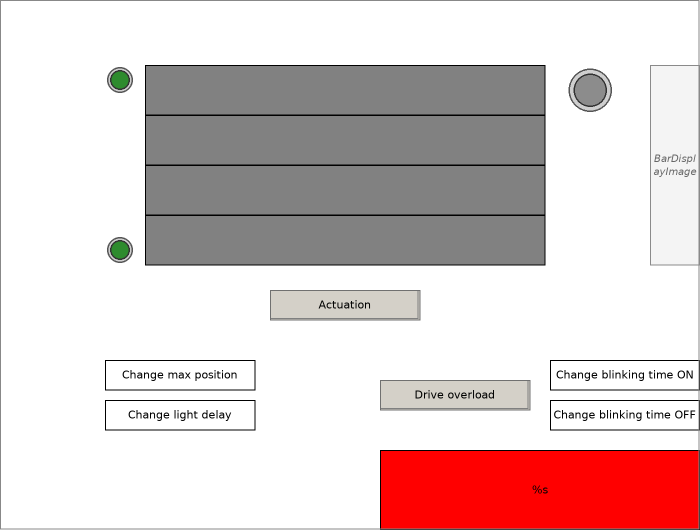
VISUALIZATION Visualization  // 700x530
    Button (270,290 150x30), "Actuation"
        tap MAIN.bActuation1
    Rectangle (145,65 400x200)
    Rectangle (145,65 400x50), invisible if: MAIN.fbGarage1.bRect4
    Rectangle (145,115 400x50), invisible if: MAIN.fbGarage1.bRect3
    Rectangle (145,165 400x50), invisible if: MAIN.fbGarage1.bRect2
    Rectangle (145,215 400x50), invisible if: MAIN.fbGarage1.bRect1
    Rectangle (105,360 150x30), "Change max position"
        OnMouseDown: write MAIN.fMaxPosition1 via Default
    Button (380,380 150x30), "Drive overload"
        tap MAIN.bDriveOverload1
    Rectangle (105,400 150x30), "Change light delay"
        OnMouseDown: write MAIN.dwLightDelay1 via Default
    Rectangle (550,360 150x30), "Change blinking time ON"
        OnMouseDown: write MAIN.dwBlinkingTimeOn1 via Default
    Rectangle (550,400 150x30), "Change blinking time OFF"
        OnMouseDown: write MAIN.dwBlinkingTimeOff1 via Default
    Rectangle (380,450 320x80), "%s", text variable: MAIN.sErrorMessage1, invisible if: MAIN.bNoError1
    Lamp1 (565,65 50x50), variable: MAIN.bDoorLight1, style: Lamp-Lamp1-Gray
    Lamp1 (105,65 30x30), variable: MAIN.bOpeningLight1, style: Lamp-Lamp1-Green
    Lamp1 (105,235 30x30), variable: MAIN.bClosingLight1, style: Lamp-Lamp1-Green
    BarDisplayImage (650,65 50x200), value: MAIN.fbGarage1.AxisGarage.NcToPlc.ActPos, style: BarDisplayImage-Gray, scale format: %.1f, scale 0..100
END_VISUALIZATION

(* stored: Version 1.1.0.1, ProductVersion 3.1.4024.12
   Visu Visualization: Id {9e447a44-0cbc-4d30-a665-e4dd7d1dbec6} *)
